// LS Electric XG5000 project: LK Tech
// PLC NewPLC

PROGRAM Main (task: 스캔 프로그램)

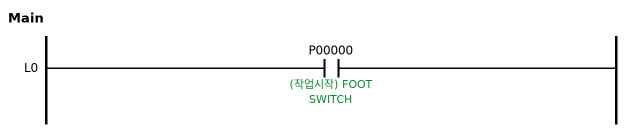
; L0
LOAD      P00000	// (작업시작) FOOT SWITCH

VARIABLES AND COMMENTS (devices not used above)
P00005	BIT	온도 컨트롤러 RELAY 출력
P00006	BIT	온도 컨트롤러 ALARM 1 출력
P00007	BIT	온도 컨트롤러 ALARM 2출력
P00008	BIT	커튼 상승 리드 센서
P00009	BIT	커튼 하강 리드 센서
P0000A	BIT	패드 상승 리드 센서
P0000B	BIT	패드 하강 리드 센서
P0000C	BIT	필름 확관 전진 센서
P0000D	BIT	필름 확관 추진 센서
P0000E	BIT	진공 전진 센서
P0000F	BIT	진공 추진 쎈서
P00010	BIT	헤드 전진 리드 센서
P00011	BIT	헤드 후진 리드 센서
P00012	BIT	헤드 상승 리드 센서
P00013	BIT	헤드 하강 리드 센서
P00014	BIT	히터 전진 리드 센서
P00015	BIT	히터 후진 리드 센서
P00016	BIT	히터 상승 리드 센서
P00017	BIT	히터 하강 리드 센서
P00018	BIT	히터 회전 리드 센서
P00019	BIT	히터 복귀 리드 센서
P00020	BIT	START LAMP
P00021	BIT	EM-STOP LAMP1
P00022	BIT	EM-STOP LAMP2
P00023	BIT	SPARE
P00024	BIT	TOWER LAMP R
P00025	BIT	TOWER LAMP Y
P00026	BIT	TOWER LAMP G
P00027	BIT	HEATER M/C
P00028	BIT	BUZZER
P00029	BIT	SPARE
P0002A	BIT	SPARE
P0002B	BIT	SPARE
P0002C	BIT	커튼 상승 하강 SOL VALVE
P0002D	BIT	패드 상승 하강 SOL VALVE
P0002E	BIT	필름 확관 전진 후진 SOL VALVE
P0002F	BIT	진공 SOL VALVE
P00030	BIT	해드 좌 우 SOL VALVE
P00034	BIT	히타 회전 SOL VALVE
P00035	BIT	이젝터 SOL VALVE
P00031	BIT	해드 상승 하강 SOL VALVE
P00032	BIT	히타 전진 후진 SOL VALVE
P00033	BIT	히타 상승 하강 SOL VALVE
P00001	BIT	(작업시작) PUSH BUTTON LAMP SWITCH
P00002	BIT	비상정지 SWITCH 1
P00003	BIT	비상정지 SWITCH 2